TYPE TL_BUSY :
(
	eTlStartUnits := 0,
	eTlCheckUnits,
	eTlSignalError
)UINT;
END_TYPE

(* stored: Version 1.1.0.1, ProductVersion 3.1.4024.2
   DUT TL_BUSY: Id {196ef372-6d38-4a30-8a23-4e8c520c63ff} *)
